FUNCTION_BLOCK CROSSCOMM_SENDER_2210DD10965A92ADC (* Service Interface Function Block Type *)
  (* Standard: 61499-2 *)
  (* Version 0.0, 9/22/2017, bababen, nxtControl GmbH, template *)
  PACKAGE Main;
  (* Compiler Cpp nxtControl builtin 1.0 *)
  {SET_ATTRIBUTE(Runtime.FBType.ImplementingType, Runtime.System#DYNGEN_CROSSCOMM_SENDER)}
  {SET_ATTRIBUTE(Configuration.GenericFBType.InterfaceParams, Runtime.System#<InterfaceList> <EventInputs> <Event Name="IND"> <With Var="VAL" /> </Event> </EventInputs> <InputVars> <VarDeclaration Name="VAL" Type="BOOL" /> </InputVars> </InterfaceList>)}
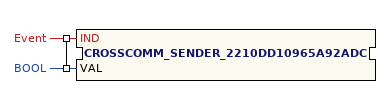
  EVENT_INPUT
    IND WITH VAL;
  END_EVENT
  VAR_INPUT
    VAL : BOOL;
  END_VAR
  EC_STATES
    START;
  END_STATES
END_FUNCTION_BLOCK
